// TIA Portal V18 export
FUNCTION_BLOCK "LED_lampTestAtStartup"   // FB43, FBD
{ S7_Optimized_Access := 'TRUE' }
VERSION : 0.1
// stored: AutoNumber true, IsIECCheckEnabled false, IsRetainMemResEnabled false, MemoryReserve 100, SetENOAutomatically false, UDAEnableTagReadback false
   VAR_IN_OUT
      HMI_TEST_ALL_LEDS : Bool;
   END_VAR
   VAR
      IEC_Timer_0_Instance { S7_SetPoint := 'True'} : TON_TIME;
      mem : Bool;
   END_VAR
   VAR_TEMP
      ton_elapsed : Bool;
      trig : Bool;
   END_VAR
   VAR_TEMP   // added for the SCL form of the ladder/FBD networks
      _w1 : Bool;
   END_VAR
BEGIN

REGION Network 1
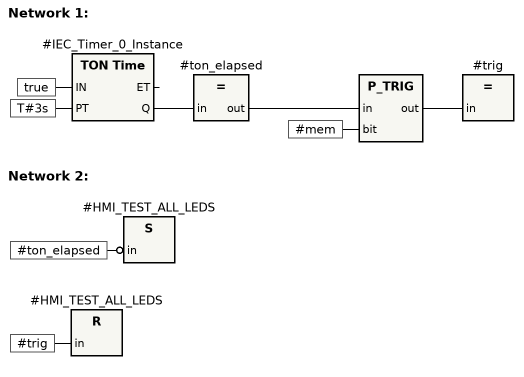
   #IEC_Timer_0_Instance(IN := true, PT := T#3s);   // TON
   #ton_elapsed := #IEC_Timer_0_Instance.Q;
   #_w1 := #IEC_Timer_0_Instance.Q AND NOT #mem;   // rising edge
   #mem := #IEC_Timer_0_Instance.Q;
   #trig := #_w1;
END_REGION

REGION Network 2
   IF NOT #ton_elapsed THEN #HMI_TEST_ALL_LEDS := TRUE; END_IF;
   IF #trig THEN #HMI_TEST_ALL_LEDS := FALSE; END_IF;
END_REGION
END_FUNCTION_BLOCK
